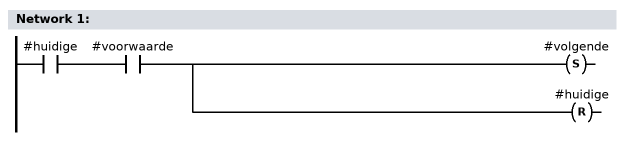
NETWORK
TITLE =
      A     #huidige;
      A     #voorwaarde;
      S     #volgende;
      R     #huidige;
END_FUNCTION

FUNCTION "Opstart_subroutine" : VOID	// FC 15
VERSION : 0.1
VAR_INPUT
  voorwaarde : BOOL ;
END_VAR
VAR_IN_OUT
  huidige : BOOL ;
  volgende_1 : BOOL ;
  volgende_2 : BOOL ;
END_VAR
BEGIN
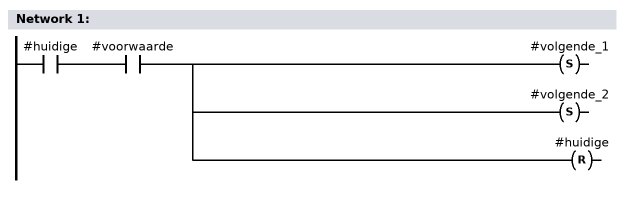
NETWORK
TITLE =
      A     #huidige;
      A     #voorwaarde;
      S     #volgende_1;
      S     #volgende_2;
      R     #huidige;
END_FUNCTION

FUNCTION "Sub_routine_gelijk" : VOID	// FC 16
VERSION : 0.1
VAR_INPUT
  voorwaarde : BOOL ;
END_VAR
VAR_IN_OUT
  huidige : BOOL ;
  volgende_1 : BOOL ;
  volgende_2 : BOOL ;
END_VAR
BEGIN
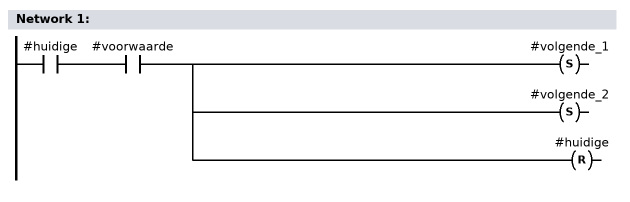
NETWORK
TITLE =
      A     #huidige;
      A     #voorwaarde;
      S     #volgende_1;
      S     #volgende_2;
      R     #huidige;
END_FUNCTION

FUNCTION "Sub_route_Station_samen" : VOID	// FC 17
VERSION : 0.1
VAR_INPUT
  voorwaarde : BOOL ;
END_VAR
VAR_IN_OUT
  huidige : BOOL ;
  volgende_1 : BOOL ;
  volgende_2 : BOOL ;
  volgende_3 : BOOL ;
END_VAR
BEGIN
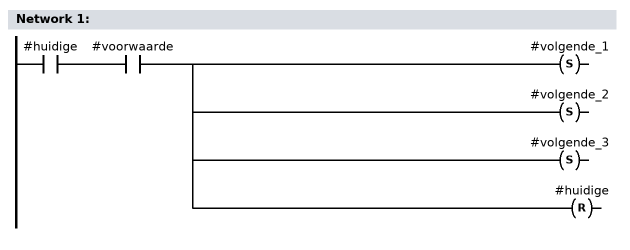
NETWORK
TITLE =
      A     #huidige;
      A     #voorwaarde;
      S     #volgende_1;
      S     #volgende_2;
      S     #volgende_3;
      R     #huidige;
END_FUNCTION

FUNCTION FC 18 : VOID
VERSION : 0.1
VAR_INPUT
  voorwaarde : BOOL ;
END_VAR
VAR_IN_OUT
  huidige_1 : BOOL ;
  huidige_2 : BOOL ;
  volgende : BOOL ;
END_VAR
BEGIN
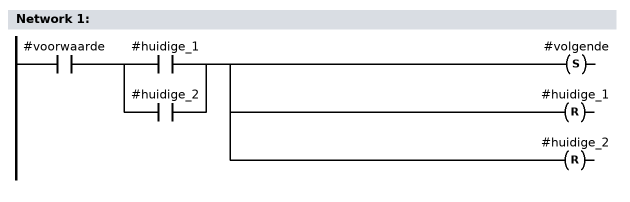
NETWORK
TITLE =
      A     #voorwaarde;
      A(;
      O     #huidige_1;
      O     #huidige_2;
      );
      S     #volgende;
      R     #huidige_1;
      R     #huidige_2;
END_FUNCTION

FUNCTION "SIM.SUBR.Y-As" : VOID	// FC 19
VERSION : 0.1
VAR_INPUT
  Balk_nr : INT ;
END_VAR
VAR_IN_OUT
  DB_Balk : INT ;
END_VAR
VAR_TEMP
  Timer2 : BOOL ;
  Timer1 : BOOL ;
  StationA : BOOL ;
  StationB : BOOL ;
END_VAR
BEGIN
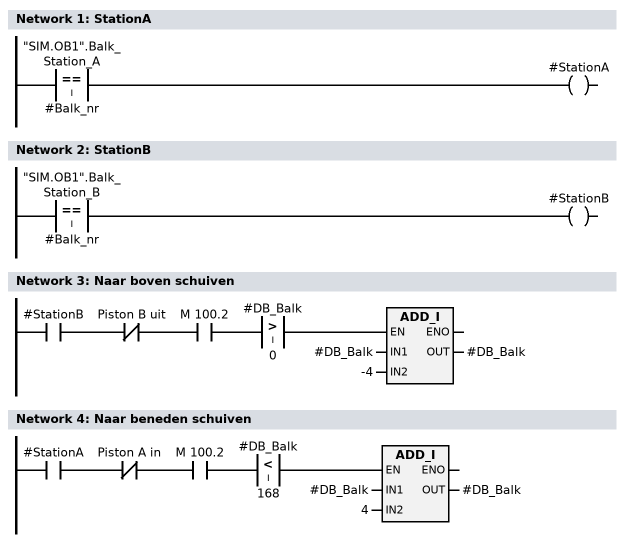
NETWORK
TITLE = StationA
      L     "SIM.OB1".Balk_Station_A;
      L     #Balk_nr;
      ==I;
      =     #StationA;
NETWORK
TITLE = StationB
      L     "SIM.OB1".Balk_Station_B;
      L     #Balk_nr;
      ==I;
      =     #StationB;
NETWORK
TITLE = Naar boven schuiven
      A     #StationB;
      AN    "Piston B uit";
      A     M 100.2;
      A(;
      L     #DB_Balk;
      L     0;
      >I;
      );
      JNB   _001;
      L     #DB_Balk;
      L     -4;
      +I;
      T     #DB_Balk;
_001: NOP   0;
NETWORK
TITLE = Naar beneden schuiven
      A     #StationA;
      AN    "Piston A in";
      A     M 100.2;
      A(;
      L     #DB_Balk;
      L     168;
      <I;
      );
      JNB   _002;
      L     #DB_Balk;
      L     4;
      +I;
      T     #DB_Balk;
_002: NOP   0;
END_FUNCTION

FUNCTION "SIM.LOGIN" : VOID	// FC 20
VERSION : 0.1
VAR_INPUT
  Login_Button : BOOL ;
  User_ID : INT ;
  User_Input : INT ;
  User_Password : DINT ;
  Password_input : DINT ;
  User_Right : INT ;
END_VAR
VAR_TEMP
  ID_OF_Input : BOOL ;
  Password_Correct : BOOL ;
END_VAR
BEGIN
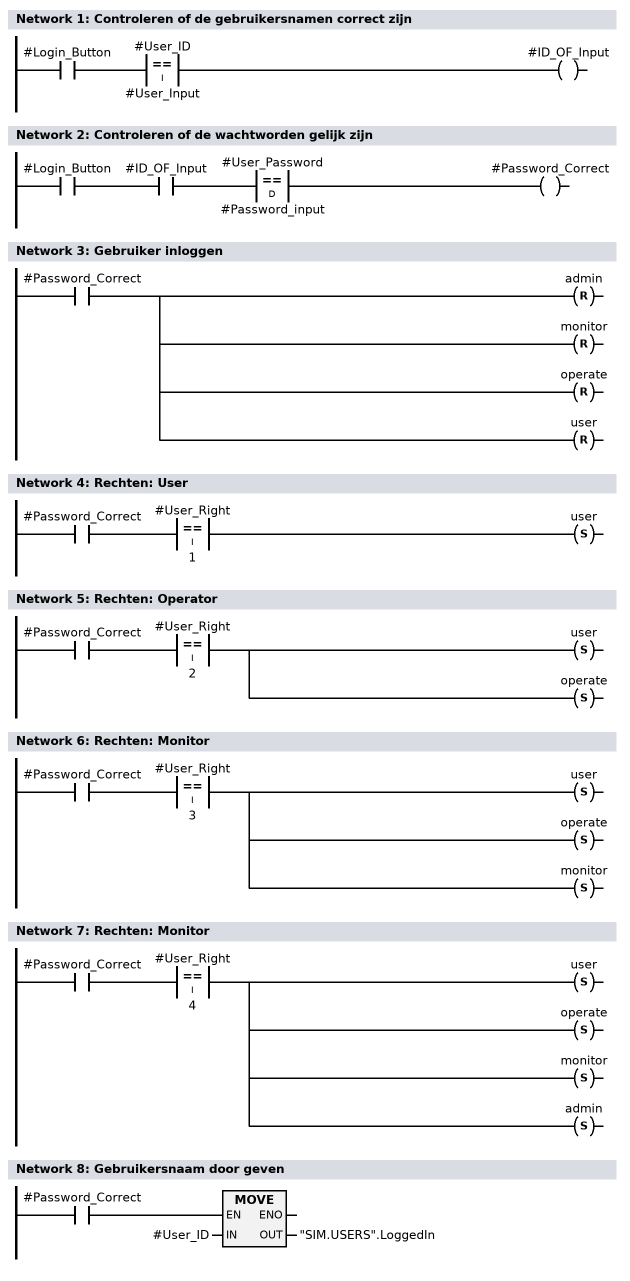
NETWORK
TITLE = Controleren of de gebruikersnamen correct zijn
      A     #Login_Button;
      A(;
      L     #User_ID;
      L     #User_Input;
      ==I;
      );
      =     #ID_OF_Input;
NETWORK
TITLE = Controleren of de wachtworden gelijk zijn
      A     #Login_Button;
      A     #ID_OF_Input;
      A(;
      L     #User_Password;
      L     #Password_input;
      ==D;
      );
      =     #Password_Correct;
NETWORK
TITLE = Gebruiker inloggen
      A     #Password_Correct;
      R     "admin";
      R     "monitor";
      R     "operate";
      R     "user";
NETWORK
TITLE = Rechten: User
      A     #Password_Correct;
      A(;
      L     #User_Right;
      L     1;
      ==I;
      );
      S     "user";
NETWORK
TITLE = Rechten: Operator
      A     #Password_Correct;
      A(;
      L     #User_Right;
      L     2;
      ==I;
      );
      S     "user";
      S     "operate";
NETWORK
TITLE = Rechten: Monitor
      A     #Password_Correct;
      A(;
      L     #User_Right;
      L     3;
      ==I;
      );
      S     "user";
      S     "operate";
      S     "monitor";
NETWORK
TITLE = Rechten: Monitor
      A     #Password_Correct;
      A(;
      L     #User_Right;
      L     4;
      ==I;
      );
      S     "user";
      S     "operate";
      S     "monitor";
      S     "admin";
NETWORK
TITLE = Gebruikersnaam door geven
      A     #Password_Correct;
      JNB   _001;
      L     #User_ID;
      T     "SIM.USERS".LoggedIn;
_001: NOP   0;
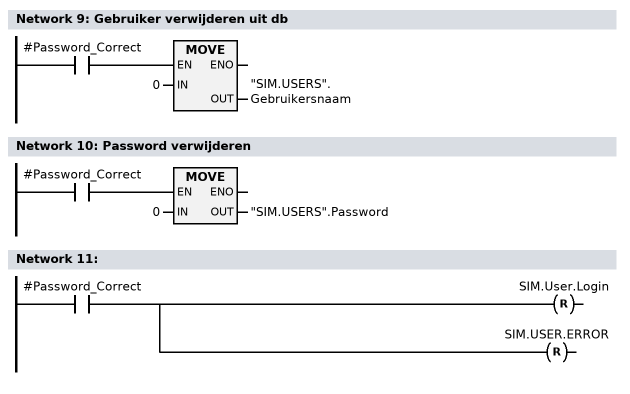
NETWORK
TITLE = Gebruiker verwijderen uit db
      A     #Password_Correct;
      JNB   _002;
      L     0;
      T     "SIM.USERS".Gebruikersnaam;
_002: NOP   0;
NETWORK
TITLE = Password verwijderen
      A     #Password_Correct;
      JNB   _003;
      L     0;
      T     "SIM.USERS".Password;
_003: NOP   0;
NETWORK
TITLE =
      A     #Password_Correct;
      R     "SIM.User.Login";
      R     "SIM.USER.ERROR";
END_FUNCTION

FUNCTION "SIM.Move.X-As" : VOID	// FC 21
VERSION : 0.1
VAR_INPUT
  Sensor : BOOL ;
  Xvalue : INT ;
END_VAR
BEGIN
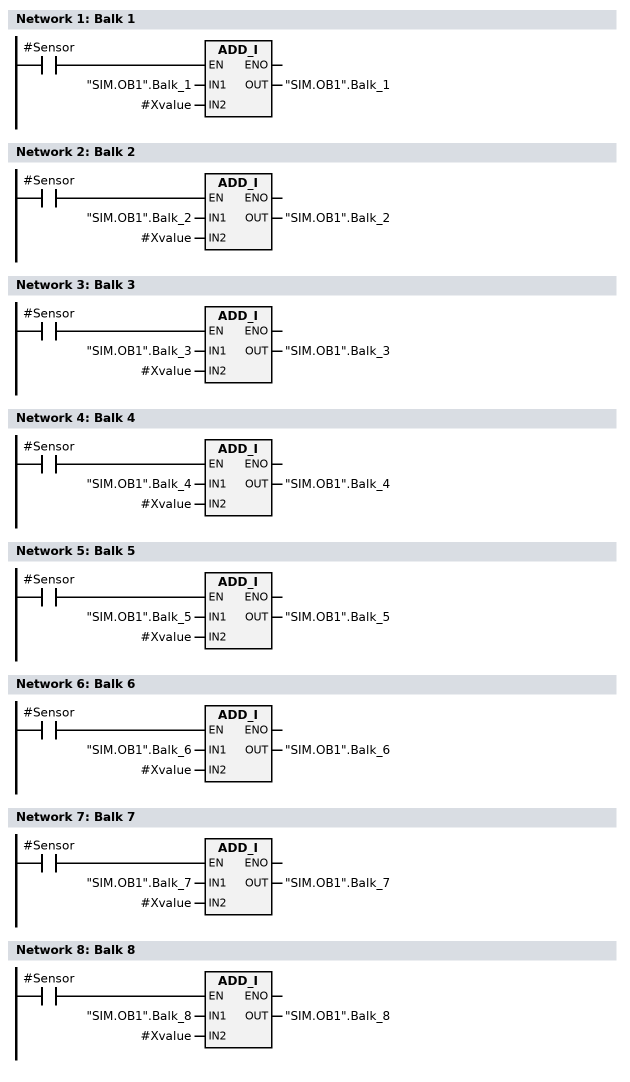
NETWORK
TITLE = Balk 1
      A     #Sensor;
      JNB   _001;
      L     "SIM.OB1".Balk_1;
      L     #Xvalue;
      +I;
      T     "SIM.OB1".Balk_1;
_001: NOP   0;
NETWORK
TITLE = Balk 2
      A     #Sensor;
      JNB   _002;
      L     "SIM.OB1".Balk_2;
      L     #Xvalue;
      +I;
      T     "SIM.OB1".Balk_2;
_002: NOP   0;
NETWORK
TITLE = Balk 3
      A     #Sensor;
      JNB   _003;
      L     "SIM.OB1".Balk_3;
      L     #Xvalue;
      +I;
      T     "SIM.OB1".Balk_3;
_003: NOP   0;
NETWORK
TITLE = Balk 4
      A     #Sensor;
      JNB   _004;
      L     "SIM.OB1".Balk_4;
      L     #Xvalue;
      +I;
      T     "SIM.OB1".Balk_4;
_004: NOP   0;
NETWORK
TITLE = Balk 5
      A     #Sensor;
      JNB   _005;
      L     "SIM.OB1".Balk_5;
      L     #Xvalue;
      +I;
      T     "SIM.OB1".Balk_5;
_005: NOP   0;
NETWORK
TITLE = Balk 6
      A     #Sensor;
      JNB   _006;
      L     "SIM.OB1".Balk_6;
      L     #Xvalue;
      +I;
      T     "SIM.OB1".Balk_6;
_006: NOP   0;
NETWORK
TITLE = Balk 7
      A     #Sensor;
      JNB   _007;
      L     "SIM.OB1".Balk_7;
      L     #Xvalue;
      +I;
      T     "SIM.OB1".Balk_7;
_007: NOP   0;
NETWORK
TITLE = Balk 8
      A     #Sensor;
      JNB   _008;
      L     "SIM.OB1".Balk_8;
      L     #Xvalue;
      +I;
      T     "SIM.OB1".Balk_8;
_008: NOP   0;
END_FUNCTION

FUNCTION "SIM.BALK.Reset" : VOID	// FC 22
VERSION : 0.1
VAR_IN_OUT
  Balk : INT ;
END_VAR
BEGIN
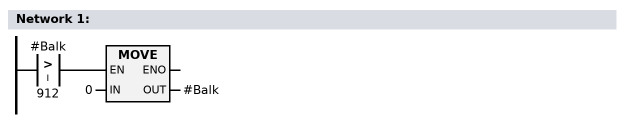
NETWORK
TITLE =
      A(;
      L     #Balk;
      L     912;
      >I;
      );
      JNB   _001;
      L     0;
      T     #Balk;
_001: NOP   0;
END_FUNCTION

FUNCTION "SUB.Posit" : VOID	// FC 23
VERSION : 0.1
VAR_INPUT
  Station : INT ;
  BalkPostitie : INT ;
  BalkNr : INT ;
  BalkMerker : BOOL ;
  Waarde : INT ;
END_VAR
VAR_OUTPUT
  ReturnStation : BOOL ;
  ActivatieStation : BOOL ;
END_VAR
VAR_TEMP
  Save : BOOL ;
END_VAR
BEGIN
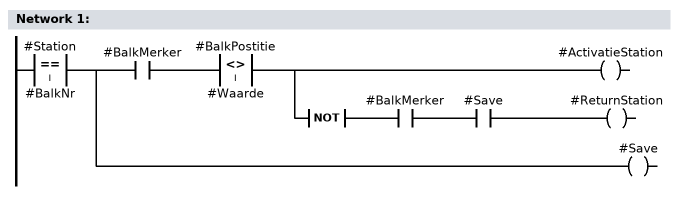
NETWORK
TITLE =
      L     #Station;
      L     #BalkNr;
      ==I;
      =     L 1.0;
      A     L 1.0;
      A     #BalkMerker;
      A(;
      L     #BalkPostitie;
      L     #Waarde;
      <>I;
      );
      =     L 1.1;
      A     L 1.1;
      BLD   102;
      =     #ActivatieStation;
      A     L 1.1;
      NOT;
      A     #BalkMerker;
      A     #Save;
      =     #ReturnStation;
      A     L 1.0;
      BLD   102;
      =     #Save;
END_FUNCTION

DATA_BLOCK DB 1
VERSION : 0.1
  STRUCT
   Ingevoerde_Waarde : INT ;
   Momentele_Waarde : INT ;
  END_STRUCT ;	
BEGIN
END_DATA_BLOCK

DATA_BLOCK "SIM.OB1"	// DB 2
VERSION : 0.1
  STRUCT
   Balk_1 : INT ;	//0
   Balk_2 : INT ;	//0
   Balk_3 : INT ;	//0
   Balk_4 : INT ;	//0
   Balk_5 : INT ;	//0
   Balk_6 : INT ;	//0
   Balk_7 : INT ;	//0
   Balk_8 : INT ;	//0
   Balk_1_boven : INT ;	//0
   Balk_2_boven : INT ;
   Balk_3_boven : INT ;
   Balk_4_boven : INT ;
   Balk_5_boven : INT ;
   Balk_6_boven : INT ;
   Balk_7_boven : INT ;
   Balk_8_boven : INT ;
   Balk_Sensoren : INT ;
   Balk_Station_A : INT ;
   Balk_Station_B : INT ;
   Balk_Station_A_Mom : INT ;	//Momentele waarde
   Balk_Station_B_Mom : INT ;	//Momentele waarde
  END_STRUCT ;	
BEGIN
END_DATA_BLOCK

DATA_BLOCK "SIM.USERS"	// DB 3
VERSION : 0.1
  STRUCT
   Gebruikersnaam : INT ;	//Temporary placeholder variable
   Password : DINT ;
   LoggedIn : INT ;
  END_STRUCT ;	
BEGIN
END_DATA_BLOCK

DATA_BLOCK "Positionering"	// DB 4
VERSION : 0.1
  STRUCT
   Balk_1 : BOOL ;	//Temporary placeholder variable
   Balk_2 : BOOL ;
   Balk_3 : BOOL ;
   Balk_4 : BOOL ;
   Balk_5 : BOOL ;
   Balk_6 : BOOL ;
   Balk_7 : BOOL ;
   Balk_8 : BOOL ;
   Recept1 : BYTE ;
   Recept2 : BYTE ;
   Recept3 : BYTE ;
   Recept4 : BYTE ;
   Recept5 : BYTE ;
   Recept6 : BYTE ;
   Recept7 : BYTE ;
   Recept8 : BYTE ;
   Recept9 : BYTE ;
   Recept10 : BYTE ;
   Recept_Save : INT ;
   Recept_Zoom : INT ;
   Return_Station_A : BOOL ;
   Return_Station_B : BOOL ;
  END_STRUCT ;	
BEGIN
END_DATA_BLOCK

ORGANIZATION_BLOCK OB 1
TITLE = "Main Program Sweep (Cycle)"
VERSION : 0.1
VAR_TEMP
  OB1_EV_CLASS : BYTE ;	//Bits 0-3 = 1 (Coming event), Bits 4-7 = 1 (Event class 1)
  OB1_SCAN_1 : BYTE ;	//1 (Cold restart scan 1 of OB 1), 3 (Scan 2-n of OB 1)
  OB1_PRIORITY : BYTE ;	//Priority of OB Execution
  OB1_OB_NUMBR : BYTE ;	//1 (Organization block 1, OB1)
  OB1_RESERVED_1 : BYTE ;	//Reserved for system
  OB1_RESERVED_2 : BYTE ;	//Reserved for system
  OB1_PREV_CYCLE : INT ;	//Cycle time of previous OB1 scan (milliseconds)
  OB1_MIN_CYCLE : INT ;	//Minimum cycle time of OB1 (milliseconds)
  OB1_MAX_CYCLE : INT ;	//Maximum cycle time of OB1 (milliseconds)
  OB1_DATE_TIME : DATE_AND_TIME ;	//Date and time OB1 started
END_VAR
BEGIN
NETWORK
TITLE =
      CALL  "Uitgangen Sturen";
      CALL  "DB_Function";
      CALL  "Timers + Counters";
      CALL  "Simulatie_Run";
      CALL  "Opstart_FC";
      CALL  "SIM.OB100";
      CALL  "SIM.user";
      CALL  "Positionering_balken";
      CALL  "Grafcet_Platform";
      CALL  "Grafcet Station A";
      CALL  "Grafcet Station B";
      CALL  "Ingang -> Merker";
END_ORGANIZATION_BLOCK

ORGANIZATION_BLOCK "COMPLETE RESTART"	// OB 100
TITLE = "Complete Restart"
VERSION : 0.1
VAR_TEMP
  OB100_EV_CLASS : BYTE ;	//16#13, Event class 1, Entering event state, Event logged in diagnostic buffer
  OB100_STRTUP : BYTE ;	//16#81/82/83/84 Method of startup
  OB100_PRIORITY : BYTE ;	//Priority of OB Execution
  OB100_OB_NUMBR : BYTE ;	//100 (Organization block 100, OB100)
  OB100_RESERVED_1 : BYTE ;	//Reserved for system
  OB100_RESERVED_2 : BYTE ;	//Reserved for system
  OB100_STOP : WORD ;	//Event that caused CPU to stop (16#4xxx)
  OB100_STRT_INFO : DWORD ;	//Information on how system started
  OB100_DATE_TIME : DATE_AND_TIME ;	//Date and time OB100 started
END_VAR
BEGIN
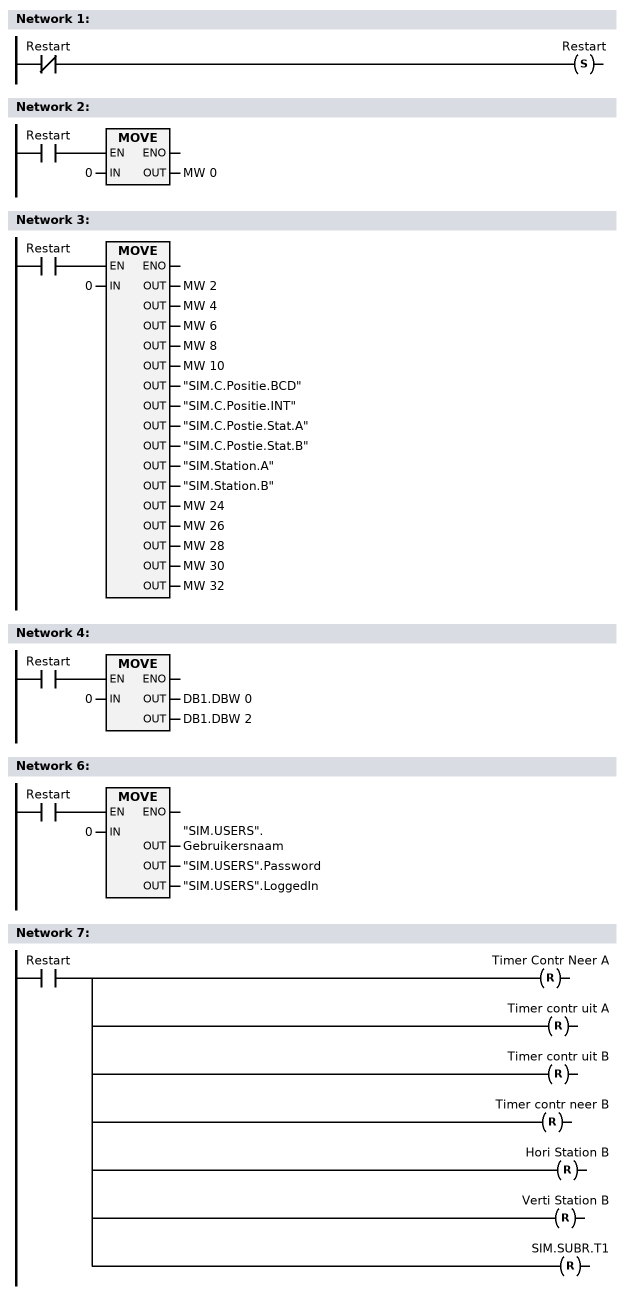
NETWORK
TITLE =
      AN    "Restart";
      S     "Restart";
NETWORK
TITLE =
      A     "Restart";
      JNB   _001;
      L     0;
      T     MW 0;
_001: NOP   0;
NETWORK
TITLE =
      A     "Restart";
      JNB   _002;
      L     0;
      T     MW 2;
      T     MW 4;
      T     MW 6;
      T     MW 8;
      T     MW 10;
      T     "SIM.C.Positie.BCD";
      T     "SIM.C.Positie.INT";
      T     "SIM.C.Postie.Stat.A";
      T     "SIM.C.Postie.Stat.B";
      T     "SIM.Station.A";
      T     "SIM.Station.B";
      T     MW 24;
      T     MW 26;
      T     MW 28;
      T     MW 30;
      T     MW 32;
_002: NOP   0;
NETWORK
TITLE =
      A     "Restart";
      JNB   _003;
      L     0;
      T     DB1.DBW 0;
      T     DB1.DBW 2;
_003: NOP   0;
NETWORK
TITLE =
      A     "Restart";
      JNB   _003;
      L     0;
      T     "SIM.OB1".Balk_1;
      T     "SIM.OB1".Balk_2;
      T     "SIM.OB1".Balk_3;
      T     "SIM.OB1".Balk_4;
      T     "SIM.OB1".Balk_5;
      T     "SIM.OB1".Balk_6;
      T     "SIM.OB1".Balk_7;
      T     "SIM.OB1".Balk_8;
      T     "SIM.OB1".Balk_1_boven;
      T     "SIM.OB1".Balk_2_boven;
      T     "SIM.OB1".Balk_3_boven;
      T     "SIM.OB1".Balk_4_boven;
      T     "SIM.OB1".Balk_5_boven;
      T     "SIM.OB1".Balk_6_boven;
      T     "SIM.OB1".Balk_7_boven;
      T     "SIM.OB1".Balk_8_boven;
NETWORK
TITLE =
      A     "Restart";
      JNB   _004;
      L     0;
      T     "SIM.USERS".Gebruikersnaam;
      T     "SIM.USERS".Password;
      T     "SIM.USERS".LoggedIn;
_004: NOP   0;
NETWORK
TITLE =
      A     "Restart";
      R     "Timer Contr Neer A";
      R     "Timer contr uit A";
      R     "Timer contr uit B";
      R     "Timer contr neer B";
      R     "Hori Station B";
      R     "Verti Station B";
      R     "SIM.SUBR.T1";
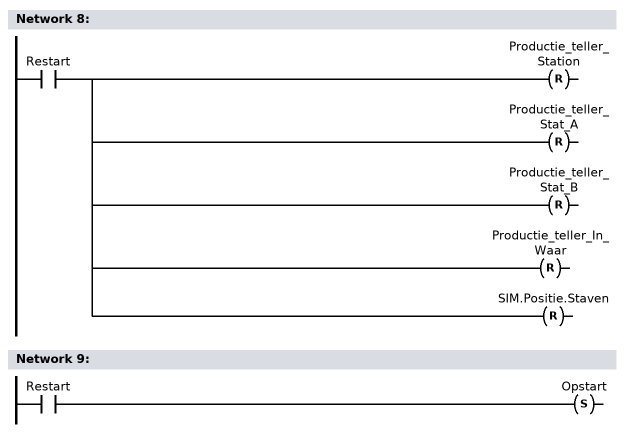
NETWORK
TITLE =
      A     "Restart";
      R     "Productie_teller_Station";
      R     "Productie_teller_Stat_A";
      R     "Productie_teller_Stat_B";
      R     "Productie_teller_In_Waar";
      R     "SIM.Positie.Staven";
NETWORK
TITLE =
      A     "Restart";
      S     "Opstart";
END_ORGANIZATION_BLOCK

SYMBOL_TABLE
"Ingangen.Doorsturen"	FC 1	FC 1
"Watchdog"	FC 2	FC 2
"Uitgangen.Prioriteit"	FC 3	FC 3
"voorbeeld"	FC 4	FC 4
"Start"	I 0.0	BOOL
"Stop"	I 0.1	BOOL
"Piston A in"	I 0.2	BOOL
"Piston A uit"	I 0.3	BOOL
"Piston A onder"	I 0.4	BOOL
"Piston A boven"	I 0.5	BOOL
"Piston B in"	I 0.6	BOOL
"Piston B uit"	I 0.7	BOOL
"Piston B onder"	I 124.0	BOOL
"Piston B boven"	I 124.1	BOOL
"Proxi Pos 1"	I 124.2	BOOL
"Proxi Pos 2"	I 124.3	BOOL
"Watch.Slave.Master.Go"	M 4.0	BOOL	// Van slave Naar Master
"Watch.Slave.Master.Back"	M 4.1	BOOL	// Van slave Naar master
"Watch.Master.Slave.Go"	M 4.2	BOOL
"Watch.Master.Slave.Back"	M 4.3	BOOL
"Watch.Slave.Sim.Go"	M 4.4	BOOL
"Watch.Slave.Sim.back"	M 4.5	BOOL
"Levens.Bit"	M 10.0	BOOL
"Levens.Bit.Fout"	M 10.1	BOOL
"Ingangen 0.x"	MB 0	BYTE
"Ingangen 124.x"	MB 1	BYTE
"Uitgangen 0.x"	MB 2	BYTE
"Uitgangen 124.x"	MB 3	BYTE
"Motor Rechts"	Q 0.1	BOOL
"Piston A Op-Neer"	Q 0.2	BOOL
"Piston A Uit-In"	Q 0.3	BOOL
"Piston B Op-Neer"	Q 0.4	BOOL
"Piston B Uit-In"	Q 0.5	BOOL
"Sign.Rood"	Q 0.6	BOOL
"Motor Links"	Q 124.0	BOOL
"Extend.proxi2"	T 0	TIMER
"Levens.bit.1"	T 1	TIMER
"Levens.bit.2"	T 2	TIMER
END_SYMBOL_TABLE
